FUNCTION_BLOCK VALUES2ARRAY_8_INT (* Service Interface Function Block Type *)
  (* Description: Copyright (c) 2014 Profactor GmbH, HR Agrartechnik GmbH This program and the accompanying materials are made available under the terms of the Eclipse Public License 2.0 which is available at https://www.eclipse.org/legal/epl-2.0/ SPDX-License-Identifier: EPL-2.0 *)
  (* Version 1.0, 2026-03-30, Franz Höpfinger, HR Agrartechnik GmbH, copy VALUES2ARRAY_2_LREAL and made this block *)
  PACKAGE eclipse4diac::convert;
  {SET_ATTRIBUTE(eclipse4diac::core::GenericClassName, 'GEN_VALUES2ARRAY')}
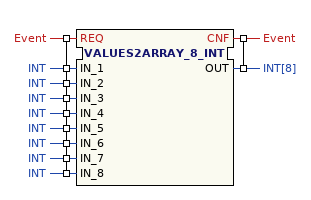
  EVENT_INPUT
    REQ WITH IN_1, IN_2, IN_3, IN_4, IN_5, IN_6, IN_7, IN_8; (* Service Request *)
  END_EVENT
  EVENT_OUTPUT
    CNF WITH OUT; (* Confirmation of Requested Service *)
  END_EVENT
  VAR_INPUT
    IN_1 : INT; (* input number 1 *)
    IN_2 : INT; (* input number 2 *)
    IN_3 : INT; (* input number 3 *)
    IN_4 : INT; (* input number 4 *)
    IN_5 : INT; (* input number 5 *)
    IN_6 : INT; (* input number 6 *)
    IN_7 : INT; (* input number 7 *)
    IN_8 : INT; (* input number 8 *)
  END_VAR
  VAR_OUTPUT
    OUT : ARRAY [0..7] OF INT; (* Array output *)
  END_VAR
END_FUNCTION_BLOCK
